# EPICS substitutions: fastFeedbackApp/Db/iocs/fbckFB05.substitutions
# File fbckFB05.substitutions
#
#
# NOTE - feedback names cannot have any spaces in them
#
# Feedback Types :
#
# define all loops here
file ../../../../db/fbckLoop.db {
  pattern { AR,  LP   ,  LN          }
          { FB05, "TR01"  , "LaunchLoop1"   }
          { FB05, "TR02"  , "LaunchLoop2"   }
          { FB05, "TR03"  , "LaunchLoop3"   }
          { FB05, "TR04"  , "LaunchLoop4"   }
          { FB05, "TR05"  , "LaunchLoop5"   }
# Every IOC will have two spares for on the fly general loop configurations
          { FB05, "GN01"  , "General1"       }
          { FB05, "GN02"  , "General2"       }
# Every IOC will have one longitudinal loop configuration
          { FB05, "LG01"  , "Longitudinal"   }
}
file ../../../../db/fbckIoc.db {
  pattern { AR }
          { FB05 }
}
